// TIA Portal V19 export
DATA_BLOCK "TEST_Production"   // DB210
// stored: MemoryReserve 100
   VAR
      O_ACT : Struct
         ABILITA_FC : Bool := FALSE;
         RETVAL : DInt := 0;
         Push : Bool := FALSE;
         Pop : Bool := FALSE;
         Pop_To_TODO : Bool := FALSE;
         Pop_To_ENDING : Bool := FALSE;
         Ordine : "Prod_Item";
      END_STRUCT;
      O_TODO : Struct
         ABILITA_FC : Bool := FALSE;
         RETVAL : DInt := 0;
         Clear_Gap : Bool := FALSE;
         Push_Top : Bool := FALSE;
         Push_Bottom : Bool := FALSE;
         Pop : Bool := FALSE;
         Pop_Index : Int;
         "Pop_&_Push_ACT" : Bool := FALSE;
         "Pop_&_Push_ENDING" : Bool := FALSE;
         Evaluate_FULL : Bool;
         Ordine : "Prod_Item";
      END_STRUCT;
      O_ENDING : Struct
         ABILITA_FC : Bool := FALSE;
         RETVAL : DInt := 0;
         Index : Int;
         Clear_Gap : Bool := FALSE;
         Push_Top : Bool := FALSE;
         Pop : Bool := FALSE;
         "Pop_&_O_OUT_Push" : Bool := FALSE;
         "Pop_&_O_TODO_Push" : Bool := FALSE;
         Ordine : "Prod_Item";
      END_STRUCT;
      O_OUT : Struct
         ABILITA_FC : Bool := FALSE;
         RETVAL : DInt := 0;
         Index : Int;
         Clear_Gap : Bool := FALSE;
         Push_Top : Bool := FALSE;
         Pop : Bool := FALSE;
         Ordine : "Prod_Item";
      END_STRUCT;
      O_ENDING_Cleaning : Struct
         Enable { ExternalAccessible := 'False'; ExternalVisible := 'False'; ExternalWritable := 'False'} : Bool;
         AckChangeStep { ExternalAccessible := 'False'; ExternalVisible := 'False'; ExternalWritable := 'False'} : Bool;
         ActualStep { ExternalAccessible := 'False'; ExternalVisible := 'False'; ExternalWritable := 'False'} : Int;
      END_STRUCT;
   END_VAR
BEGIN
   O_ACT.Ordine.O_ID := 567;
   O_ACT.Ordine."Type" := 1;
   O_ACT.Ordine.Status := 0;
   O_ACT.Ordine.Status_Saved := 0;
   O_ACT.Ordine.Material_Len_REQ := 1997501.0;
   O_ACT.Ordine.Material_Len_ToGo := 1997501.0;
   O_ACT.Ordine.MES_IDP := 'Test MSG100';
   O_ACT.Ordine.MES_Profile_Code := 'C';
   O_ACT.Ordine.MES_PPrf_Name := 'C060x45x1.25';
   O_ACT.Ordine.PPrf_No := 200;
   O_ACT.Ordine.Beam_Code := 0;
   O_ACT.Ordine.Beams_W_A := 45.0;
   O_ACT.Ordine.Beams_H_B := 60.0;
   O_ACT.Ordine.Beams_Thickness := 1.25;
   O_ACT.Ordine.Beams_Len_Min := 1999.0;
   O_ACT.Ordine.Beams_Len_Max := 2000.0;
   O_ACT.Ordine.Beams_Len := 2000.0;
   O_ACT.Ordine.Beams_REQ := 999;
   O_ACT.Ordine.Beams_ToGo := 999;
   O_ACT.Ordine.Beams_NonConforming := 0;
   O_ACT.Ordine.Beams_GOOD := 0;
   O_ACT.Ordine.Beams_GOOD_R := 0;
   O_ACT.Ordine.Beams_NG := 0;
   O_ACT.Ordine.Beams_TOCHECK := 0;
   O_ACT.Ordine.Parts_Len := 1999.5;
   O_ACT.Ordine.Parts_Tol := 0.5;
   O_ACT.Ordine.Parts_REQ := 999;
   O_ACT.Ordine.Parts_ToGo := 999;
   O_ACT.Ordine.Parts_NonConforming := 0;
   O_ACT.Ordine.Parts_GOOD := 0;
   O_ACT.Ordine.Parts_GOOD_R := 0;
   O_ACT.Ordine.Parts_NG := 0;
   O_ACT.Ordine.Parts_TOCHECK := 0;
   O_ACT.Ordine.Kanban_Style := FALSE;
   O_ACT.Ordine.Use_Ribbing_Roll := FALSE;
   O_ACT.Ordine.Use_Trace_Mark_Tool := FALSE;
   O_ACT.Ordine.Use_Thick_Mark_Tool := FALSE;
   O_ACT.Ordine.PackLayout_BeamsPerLayer := 10;
   O_ACT.Ordine.PackLayout_Layers_Qty := 5;
   O_TODO.Ordine.O_ID := 0;
   O_TODO.Ordine."Type" := 1;
   O_TODO.Ordine.Status := 0;
   O_TODO.Ordine.Status_Saved := 0;
   O_TODO.Ordine.Material_Len_REQ := 1997501.0;
   O_TODO.Ordine.Material_Len_ToGo := 1997501.0;
   O_TODO.Ordine.MES_IDP := 'Test MSG100';
   O_TODO.Ordine.MES_Profile_Code := 'C';
   O_TODO.Ordine.MES_PPrf_Name := 'C060x45x1.25';
   O_TODO.Ordine.PPrf_No := 1;
   O_TODO.Ordine.Beam_Code := 0;
   O_TODO.Ordine.Beams_W_A := 45.0;
   O_TODO.Ordine.Beams_H_B := 60.0;
   O_TODO.Ordine.Beams_Thickness := 1.25;
   O_TODO.Ordine.Beams_Len_Min := 1999.0;
   O_TODO.Ordine.Beams_Len_Max := 2000.0;
   O_TODO.Ordine.Beams_Len := 2000.0;
   O_TODO.Ordine.Beams_REQ := 999;
   O_TODO.Ordine.Beams_ToGo := 999;
   O_TODO.Ordine.Beams_NonConforming := 0;
   O_TODO.Ordine.Beams_GOOD := 0;
   O_TODO.Ordine.Beams_GOOD_R := 0;
   O_TODO.Ordine.Beams_NG := 0;
   O_TODO.Ordine.Beams_TOCHECK := 0;
   O_TODO.Ordine.Parts_Len := 1999.5;
   O_TODO.Ordine.Parts_Tol := 0.5;
   O_TODO.Ordine.Parts_REQ := 999;
   O_TODO.Ordine.Parts_ToGo := 999;
   O_TODO.Ordine.Parts_NonConforming := 0;
   O_TODO.Ordine.Parts_GOOD := 0;
   O_TODO.Ordine.Parts_GOOD_R := 0;
   O_TODO.Ordine.Parts_NG := 0;
   O_TODO.Ordine.Parts_TOCHECK := 0;
   O_TODO.Ordine.Kanban_Style := FALSE;
   O_TODO.Ordine.Use_Ribbing_Roll := FALSE;
   O_TODO.Ordine.Use_Trace_Mark_Tool := FALSE;
   O_TODO.Ordine.Use_Thick_Mark_Tool := FALSE;
   O_TODO.Ordine.PackLayout_BeamsPerLayer := 10;
   O_TODO.Ordine.PackLayout_Layers_Qty := 5;
   O_ENDING.Ordine.O_ID := 555;
   O_ENDING.Ordine."Type" := 1;
   O_ENDING.Ordine.Status := 0;
   O_ENDING.Ordine.Status_Saved := 0;
   O_ENDING.Ordine.Material_Len_REQ := 1997501.0;
   O_ENDING.Ordine.Material_Len_ToGo := 1997501.0;
   O_ENDING.Ordine.MES_IDP := 'Test MSG100';
   O_ENDING.Ordine.MES_Profile_Code := 'C';
   O_ENDING.Ordine.MES_PPrf_Name := 'C060x45x1.25';
   O_ENDING.Ordine.PPrf_No := 1;
   O_ENDING.Ordine.Beam_Code := 0;
   O_ENDING.Ordine.Beams_W_A := 45.0;
   O_ENDING.Ordine.Beams_H_B := 60.0;
   O_ENDING.Ordine.Beams_Thickness := 1.25;
   O_ENDING.Ordine.Beams_Len_Min := 1999.0;
   O_ENDING.Ordine.Beams_Len_Max := 2000.0;
   O_ENDING.Ordine.Beams_Len := 2000.0;
   O_ENDING.Ordine.Beams_REQ := 999;
   O_ENDING.Ordine.Beams_ToGo := 999;
   O_ENDING.Ordine.Beams_NonConforming := 0;
   O_ENDING.Ordine.Beams_GOOD := 0;
   O_ENDING.Ordine.Beams_GOOD_R := 0;
   O_ENDING.Ordine.Beams_NG := 0;
   O_ENDING.Ordine.Beams_TOCHECK := 0;
   O_ENDING.Ordine.Parts_Len := 1999.5;
   O_ENDING.Ordine.Parts_Tol := 0.5;
   O_ENDING.Ordine.Parts_REQ := 999;
   O_ENDING.Ordine.Parts_ToGo := 999;
   O_ENDING.Ordine.Parts_NonConforming := 0;
   O_ENDING.Ordine.Parts_GOOD := 0;
   O_ENDING.Ordine.Parts_GOOD_R := 0;
   O_ENDING.Ordine.Parts_NG := 0;
   O_ENDING.Ordine.Parts_TOCHECK := 0;
   O_ENDING.Ordine.Kanban_Style := FALSE;
   O_ENDING.Ordine.Use_Ribbing_Roll := FALSE;
   O_ENDING.Ordine.Use_Trace_Mark_Tool := FALSE;
   O_ENDING.Ordine.Use_Thick_Mark_Tool := FALSE;
   O_ENDING.Ordine.PackLayout_BeamsPerLayer := 10;
   O_ENDING.Ordine.PackLayout_Layers_Qty := 5;
   O_OUT.Ordine.O_ID := 555;
   O_OUT.Ordine."Type" := 1;
   O_OUT.Ordine.Status := 0;
   O_OUT.Ordine.Status_Saved := 0;
   O_OUT.Ordine.Material_Len_REQ := 1997501.0;
   O_OUT.Ordine.Material_Len_ToGo := 1997501.0;
   O_OUT.Ordine.MES_IDP := 'Test MSG100';
   O_OUT.Ordine.MES_Profile_Code := 'C';
   O_OUT.Ordine.MES_PPrf_Name := 'C060x45x1.25';
   O_OUT.Ordine.PPrf_No := 1;
   O_OUT.Ordine.Beam_Code := 0;
   O_OUT.Ordine.Beams_W_A := 45.0;
   O_OUT.Ordine.Beams_H_B := 60.0;
   O_OUT.Ordine.Beams_Thickness := 1.25;
   O_OUT.Ordine.Beams_Len_Min := 1999.0;
   O_OUT.Ordine.Beams_Len_Max := 2000.0;
   O_OUT.Ordine.Beams_Len := 2000.0;
   O_OUT.Ordine.Beams_REQ := 999;
   O_OUT.Ordine.Beams_ToGo := 999;
   O_OUT.Ordine.Beams_NonConforming := 0;
   O_OUT.Ordine.Beams_GOOD := 0;
   O_OUT.Ordine.Beams_GOOD_R := 0;
   O_OUT.Ordine.Beams_NG := 0;
   O_OUT.Ordine.Beams_TOCHECK := 0;
   O_OUT.Ordine.Parts_Len := 1999.5;
   O_OUT.Ordine.Parts_Tol := 0.5;
   O_OUT.Ordine.Parts_REQ := 999;
   O_OUT.Ordine.Parts_ToGo := 999;
   O_OUT.Ordine.Parts_NonConforming := 0;
   O_OUT.Ordine.Parts_GOOD := 0;
   O_OUT.Ordine.Parts_GOOD_R := 0;
   O_OUT.Ordine.Parts_NG := 0;
   O_OUT.Ordine.Parts_TOCHECK := 0;
   O_OUT.Ordine.Kanban_Style := FALSE;
   O_OUT.Ordine.Use_Ribbing_Roll := FALSE;
   O_OUT.Ordine.Use_Trace_Mark_Tool := FALSE;
   O_OUT.Ordine.Use_Thick_Mark_Tool := FALSE;
   O_OUT.Ordine.PackLayout_BeamsPerLayer := 10;
   O_OUT.Ordine.PackLayout_Layers_Qty := 5;
END_DATA_BLOCK
